(*			
	RafalOS
	Rafał Osajda		12.11.2025		TC 4024.66
	Zbiór metod umożliwiające odczyt danych z hmi 
*)
INTERFACE ITF_HMIEButton_HMI_Connector EXTENDS ITF_BaseComponent_HMI_Connector

END_INTERFACE

(* stored: Version 1.1.0.1
   Itf ITF_HMIEButton_HMI_Connector: Id {844b6e15-1809-0471-0178-ea9b0092663b} *)
